// TIA Portal V17 export
// export: Created 2024-09-02T12:50:40.7687317Z, ExportSetting WithDefaults, DisplayName Totally Integrated Automation Portal, DisplayVersion V17, DisplayName TIA Portal Openness, DisplayVersion V17, DisplayName TIA Portal Version Control Interface, DisplayVersion V17, DisplayName STEP 7 Professional, DisplayVersion V17, DisplayName STEP 7 Safety, DisplayVersion V17, DisplayName WinCC Professional, DisplayVersion V17
TYPE "Aveva_Data_Result"
// stored: IsFailsafeCompliant false
   STRUCT
      General_Info : "Aveva_Result_General_info";   // General information for all Station
      Global_Result_Station { S7_SetPoint := 'True'} : "Aveva_Result_Global_Result_Station";
   END_STRUCT;
END_TYPE
